{attribute 'qualified_only'}
VAR_GLOBAL
	frontend : ST_Frontend;
END_VAR

(* stored: Version 1.1.0.1
   GVL GVL_Exchange: Id {d2863a7c-52b3-4c35-8128-b55e014182d7} *)
